(*

## Short summary
An abstract CycleManager implementation to provide basic functionality.
Does not update the state of the cyclemanager, it only provides some protected update functions.

.. <info>
If used in the same step, the order/precedence of method calls should be like this:
configurations
enter
executeCommand
evaluate
waitFor
proceed
proceedWith
acknowledge
leave
.. </info>

.. <legal notes>

legal notes
=================
| SPDX-FileCopyrightText: © 2024 ekvip automation GmbH <info@ekvip.de>
| SPDX-License-Identifier: Apache-2.0
| For details check: Apache-2.0_

.. _Apache-2.0: https://www.apache.org/licenses/LICENSE-2.0

.. </legal notes>



*)
FUNCTION_BLOCK ABSTRACT AbstractCycleManager 
EXTENDS CNM_AssertionInterfaces.AbstractAssertor 
IMPLEMENTS CNM_CycleManagerInterfaces.ISingleExecutionCycleManager, 
	CNM_CycleManagerInterfaces.ICycleManagerDefaultParameters, 
	ICycleManagerStepParameters
//config
VAR
	sequenceErrorStep :DINT := STEP_ERROR;
	sequencePauseEnabled :BOOL := FALSE;
	sequenceSteppingEnabled :BOOL := FALSE;
	sequenceTimeOut :TIME := T#0S;
	sequenceStopRequestMode :CNM_CycleManagerInterfaces.StepStopRequestMode := CNM_CycleManagerInterfaces.StepStopRequestMode.IGNORE;
	sequenceTimeoutStep :DINT := STEP_ERROR;
	sequenceStepWidth :DINT := 1;
	sequenceRequireSuccessStep :BOOL := FALSE;
	
	stepErrorStep :DINT := STEP_ERROR;
	stepPauseEnabled :BOOL := FALSE;
	stepSteppingEnabled :BOOL := FALSE;
	stepTimeOut :TIME := T#0S;
	stepCurrentStopRequestMode :CNM_CycleManagerInterfaces.StepStopRequestMode := CNM_CycleManagerInterfaces.StepStopRequestMode.IGNORE;
	stepTimeoutStep :DINT := STEP_ERROR;
	stepStepWidth :DINT := 1;
END_VAR
VAR
	lastStepBeforePause : DINT;
	lastStep : DINT;
	
	currentStep : DINT := CNM_ReturnTypes.DefaultSteps.STEP.IDLE;
	nextStep : DINT := CNM_ReturnTypes.DefaultSteps.STEP.IDLE;
	nextStepSpecifiedByUser :BOOL := FALSE;
	lastExecute : BOOL;
	externalExecute : BOOL;
	currentState : CNM_ReturnTypes.SingleExecutionState := CNM_ReturnTypes.SingleExecutionState.IDLE;
	wasError : BOOL;
	wasTimeoutError : BOOL;
	gotHereByError : BOOL;
	stepLastCycle : DINT;
	wasNotSuccess: BOOL;
	wasSuccess: BOOL;
	firstCycle : BOOL;
	timeoutTimer : TON;
	
	//used for cycle time optimizations
	registeredEnter : BOOL;
	registeredCommand : BOOL;
	registeredEval : BOOL;
	registeredLeave : BOOL;	
END_VAR
VAR CONSTANT
	STEP_IDLE :DINT := CNM_ReturnTypes.DefaultSteps.STEP.IDLE;
	STEP_INIT :DINT := CNM_ReturnTypes.DefaultSteps.STEP.INIT;
	STEP_ERROR :DINT := CNM_ReturnTypes.DefaultSteps.STEP.ERROR;
	STEP_ABORT :DINT := CNM_ReturnTypes.DefaultSteps.STEP.ABORT;
	STEP_PAUSE :DINT := CNM_ReturnTypes.DefaultSteps.STEP.PAUSE;
	STEP_SUCCESS :DINT := CNM_ReturnTypes.DefaultSteps.STEP.SUCCESS;	
END_VAR


(*

## Short summary
This method acknowledges an error in the state machine and resets the current step to the step befor the error occured.

.. <legal notes>

legal notes
=================
| SPDX-FileCopyrightText: © 2024 ekvip automation GmbH <info@ekvip.de>
| SPDX-License-Identifier: Apache-2.0
| For details check: Apache-2.0_

.. _Apache-2.0: https://www.apache.org/licenses/LICENSE-2.0

.. </legal notes>

*)
{attribute 'hide'}
METHOD acknowledge
IF(THIS^.gotHereByError)THEN
	THIS^.next := THIS^.last;
	THIS^.wasNotSuccess := FALSE;
	THIS^.wasError := FALSE;
	THIS^.wasTimeoutError := FALSE;
	THIS^.wasSuccess := TRUE;
END_IF
END_METHOD

(*

## Short summary
This method is called if an assertion was ``FALSE``

.. <legal notes>

legal notes
=================
| SPDX-FileCopyrightText: © 2022 ekvip automation GmbH <info@ekvip.de>
| SPDX-License-Identifier: Apache-2.0
| For details check: Apache-2.0_

.. _Apache-2.0: https://www.apache.org/licenses/LICENSE-2.0

.. </legal notes>


*)
METHOD assertionWasWrong
VAR_INPUT
	(* caller object of the method *)
	caller	: CNM_AbstractObject.IObject;
	(* alarm message *)
	message	: CNM_AssertionInterfaces.AssertMessage;
	(* debugging information *)
	additionalText	: Tc2_System.T_MaxString;
END_VAR
THIS^.wasError := TRUE;
THIS^.wasSuccess := FALSE;
THIS^.wasNotSuccess := TRUE;
END_METHOD

(*

## Short summary
An interface to provide configurations for cycle manager in a fluent way.

.. <legal notes>

legal notes
=================
| SPDX-FileCopyrightText: © 2024 ekvip automation GmbH <info@ekvip.de>
| SPDX-License-Identifier: Apache-2.0
| For details check: Apache-2.0_

.. _Apache-2.0: https://www.apache.org/licenses/LICENSE-2.0

.. </legal notes>



*)
PROPERTY configuration : CNM_CycleManagerInterfaces.ICycleManagerConfigurationScope
GET
VAR_INST
	configurator :CycleManagerConfigurator(THIS^, THIS^);
END_VAR
configuration := configurator;
END_GET
END_PROPERTY

(*

## Short summary
This property returns the current step of the cycle manager.
Proposed use is as CASE control.

### Example
```
CASE cyclemanager.steps.current OF
DefaultSteps.STEP.IDLE:
	;
DefaultSteps.STEP.INIT:
	;
2:
	;
3:
	;
4:
	;
DefaultSteps.STEP.SUCCESS:
	;
DefaultSteps.STEP.ERROR:
	;
DefaultSteps.STEP.ABORT:
	;
ELSE ;
END_CASE
```

.. <legal notes>

legal notes
=================
| SPDX-FileCopyrightText: © 2024 ekvip automation GmbH <info@ekvip.de>
| SPDX-License-Identifier: Apache-2.0
| For details check: Apache-2.0_

.. _Apache-2.0: https://www.apache.org/licenses/LICENSE-2.0

.. </legal notes>

*)
{attribute 'hide'}
PROPERTY current : DINT
GET
current := THIS^.currentStep;
END_GET
SET // PRIVATE
THIS^.currentStep := current;
END_SET
END_PROPERTY

{attribute 'hide'}
PROPERTY currentErrorStep : DINT
GET // PROTECTED
currentErrorStep := THIS^.stepErrorStep;
END_GET
SET
THIS^.stepErrorStep := currentErrorStep;
END_SET
END_PROPERTY

{attribute 'hide'}
PROPERTY currentPauseEnabled : BOOL
GET // PROTECTED
currentPauseEnabled := THIS^.stepPauseEnabled;
END_GET
SET
THIS^.stepPauseEnabled := currentPauseEnabled;
END_SET
END_PROPERTY

{attribute 'hide'}
PROPERTY currentSteppingEnabled : BOOL
GET // PROTECTED
currentSteppingEnabled := THIS^.stepSteppingEnabled;
END_GET
SET
THIS^.stepSteppingEnabled := currentSteppingEnabled;
END_SET
END_PROPERTY

{attribute 'hide'}
PROPERTY currentStepWidth : DINT
GET // PROTECTED
currentStepWidth := THIS^.stepStepWidth;
END_GET
SET
THIS^.stepStepWidth := currentStepWidth;
END_SET
END_PROPERTY

{attribute 'hide'}
PROPERTY currentStopRequestMode : CNM_CycleManagerInterfaces.StepStopRequestMode
GET // PROTECTED
currentStopRequestMode := THIS^.stepCurrentStopRequestMode;
END_GET
SET
THIS^.stepCurrentStopRequestMode := currentStopRequestMode;
END_SET
END_PROPERTY

(*

## Short summary
This property sets the maximum execution time for the current step. 
The cycle manager will go into the error step after the time elapsed.

.. <legal notes>

legal notes
=================
| SPDX-FileCopyrightText: © 2024 ekvip automation GmbH <info@ekvip.de>
| SPDX-License-Identifier: Apache-2.0
| For details check: Apache-2.0_

.. _Apache-2.0: https://www.apache.org/licenses/LICENSE-2.0

.. </legal notes>

*)
{attribute 'hide'}
PROPERTY currentTimeout : TIME
GET // PROTECTED
currentTimeout := THIS^.stepTimeOut;
END_GET
SET
THIS^.stepTimeOut := currentTimeout;
END_SET
END_PROPERTY

{attribute 'hide'}
PROPERTY currentTimeoutStep : DINT
GET // PROTECTED
IF(THIS^.stepTimeoutStep <> THIS^.defaultTimeoutStep OR THIS^.stepTimeoutStep <> THIS^.defaultErrorStep)THEN
	currentTimeoutStep := THIS^.stepTimeoutStep;	
ELSE
	currentTimeoutStep := THIS^.currentErrorStep;
END_IF
END_GET
SET
THIS^.stepTimeoutStep := currentTimeoutStep;
END_SET
END_PROPERTY

(*

## Short summary
This property stes the next step in case of an error after a step change.

.. <legal notes>

legal notes
=================
| SPDX-FileCopyrightText: © 2024 ekvip automation GmbH <info@ekvip.de>
| SPDX-License-Identifier: Apache-2.0
| For details check: Apache-2.0_

.. _Apache-2.0: https://www.apache.org/licenses/LICENSE-2.0

.. </legal notes>

*)

{attribute 'hide'}
PROPERTY defaultErrorStep : DINT
GET // PROTECTED
defaultErrorStep := THIS^.sequenceErrorStep;
END_GET
SET
THIS^.sequenceErrorStep := defaultErrorStep;
THIS^.currentErrorStep := defaultErrorStep;
END_SET
END_PROPERTY

(*

## Short summary
This property sets the default pause enabling state after a step change.

.. <legal notes>

legal notes
=================
| SPDX-FileCopyrightText: © 2024 ekvip automation GmbH <info@ekvip.de>
| SPDX-License-Identifier: Apache-2.0
| For details check: Apache-2.0_

.. _Apache-2.0: https://www.apache.org/licenses/LICENSE-2.0

.. </legal notes>

*)

{attribute 'hide'}
PROPERTY defaultPauseEnabled : BOOL
GET // PROTECTED
defaultPauseEnabled := THIS^.sequencePauseEnabled;
END_GET
SET
THIS^.sequencePauseEnabled := defaultPauseEnabled;
THIS^.currentPauseEnabled := defaultPauseEnabled;
END_SET
END_PROPERTY

(*

## Short summary
Specifies whether the SUCCESS step of the state machine can be skipped when the transition condition to SUCCESS is already fulfilled.

When set to false, the state machine immediately returns SUCCESS as soon as the transition condition to the SUCCESS state is met, 
without executing the dedicated SUCCESS step. This optimization can save one execution cycle per state machine invocation, which is 
especially beneficial in nested or complex state machine structures.

When set to true, the SUCCESS step will always be executed at least once before the state machine returns SUCCESS. This is required 
in cases where the SUCCESS step performs essential actions (e.g., resetting outputs, logging, or cleanup).

The default value is false.

Use Case:
Use false when the SUCCESS step has no functional side effects and skipping it can improve performance.
Use true when the SUCCESS step contains logic that must be executed explicitly.

.. <legal notes>

legal notes
=================
| SPDX-FileCopyrightText: © 2025 ekvip automation GmbH <info@ekvip.de>
| SPDX-License-Identifier: Apache-2.0
| For details check: Apache-2.0_

.. _Apache-2.0: https://www.apache.org/licenses/LICENSE-2.0

.. </legal notes>

*)

PROPERTY defaultRequireSuccessStep : BOOL
GET
defaultRequireSuccessStep := THIS^.sequenceRequireSuccessStep;
END_GET
SET
THIS^.sequenceRequireSuccessStep := defaultRequireSuccessStep;
END_SET
END_PROPERTY

(*

## Short summary
This property sets the default stepping mode configuration after a step change.

.. <legal notes>

legal notes
=================
| SPDX-FileCopyrightText: © 2024 ekvip automation GmbH <info@ekvip.de>
| SPDX-License-Identifier: Apache-2.0
| For details check: Apache-2.0_

.. _Apache-2.0: https://www.apache.org/licenses/LICENSE-2.0

.. </legal notes>

*)

{attribute 'hide'}
PROPERTY defaultSteppingEnabled : BOOL
GET // PROTECTED
defaultSteppingEnabled := THIS^.sequenceSteppingEnabled;
END_GET
SET
THIS^.sequenceSteppingEnabled := defaultSteppingEnabled;
THIS^.currentSteppingEnabled := defaultSteppingEnabled;
END_SET
END_PROPERTY

(*

## Short summary
This property sets the default the step width.

.. <legal notes>

legal notes
=================
| SPDX-FileCopyrightText: © 2024 ekvip automation GmbH <info@ekvip.de>
| SPDX-License-Identifier: Apache-2.0
| For details check: Apache-2.0_

.. _Apache-2.0: https://www.apache.org/licenses/LICENSE-2.0

.. </legal notes>

*)

{attribute 'hide'}
PROPERTY defaultStepWidth : DINT
GET // PROTECTED
defaultStepWidth := THIS^.sequenceStepWidth;
END_GET
SET
THIS^.sequenceStepWidth := defaultStepWidth;
THIS^.currentStepWidth := defaultStepWidth;
END_SET
END_PROPERTY

(*

## Short summary
This property sets the default step mode configuration. 

.. <legal notes>

legal notes
=================
| SPDX-FileCopyrightText: © 2024 ekvip automation GmbH <info@ekvip.de>
| SPDX-License-Identifier: Apache-2.0
| For details check: Apache-2.0_

.. _Apache-2.0: https://www.apache.org/licenses/LICENSE-2.0

.. </legal notes>

*)

{attribute 'hide'}
PROPERTY defaultStopRequestMode : CNM_CycleManagerInterfaces.StepStopRequestMode
GET // PROTECTED
defaultStopRequestMode := THIS^.sequenceStopRequestMode;
END_GET
SET
THIS^.sequenceStopRequestMode := defaultStopRequestMode;
THIS^.currentStopRequestMode := defaultStopRequestMode;
END_SET
END_PROPERTY

(*

## Short summary
This property sets the maximum execution time for steps. 
The cycle manager will go into the timeoutStep after the time elapsed.

.. <legal notes>

legal notes
=================
| SPDX-FileCopyrightText: © 2024 ekvip automation GmbH <info@ekvip.de>
| SPDX-License-Identifier: Apache-2.0
| For details check: Apache-2.0_

.. _Apache-2.0: https://www.apache.org/licenses/LICENSE-2.0

.. </legal notes>

*)

{attribute 'hide'}
PROPERTY defaultTimeout : TIME
GET // PROTECTED
defaultTimeout := THIS^.sequenceTimeOut;
END_GET
SET
THIS^.sequenceTimeOut := defaultTimeout;
THIS^.currentTimeout := defaultTimeout;
END_SET
END_PROPERTY

(*

## Short summary
This property sets the default step that will be set if the current step reaches a timeout. 

.. <legal notes>

legal notes
=================
| SPDX-FileCopyrightText: © 2024 ekvip automation GmbH <info@ekvip.de>
| SPDX-License-Identifier: Apache-2.0
| For details check: Apache-2.0_

.. _Apache-2.0: https://www.apache.org/licenses/LICENSE-2.0

.. </legal notes>

*)

{attribute 'hide'}
PROPERTY defaultTimeoutStep : DINT
GET // PROTECTED
defaultTimeoutStep := THIS^.sequenceTimeoutStep;
END_GET
SET
THIS^.sequenceTimeoutStep := defaultTimeoutStep;
THIS^.currentTimeoutStep := defaultTimeoutStep;
END_SET
END_PROPERTY

(*

## Short summary
This method performs the given invoke only in the first cycle of the current step.

.. <legal notes>

legal notes
=================
| SPDX-FileCopyrightText: © 2024 ekvip automation GmbH <info@ekvip.de>
| SPDX-License-Identifier: Apache-2.0
| For details check: Apache-2.0_

.. _Apache-2.0: https://www.apache.org/licenses/LICENSE-2.0

.. </legal notes>


*)
METHOD enter
VAR_INPUT
	(* command to execute *)
	invoke	:CNM_CommandInterfaces.ISingleAttempt;
	(* step to proceed with in case of error *)
	errorStep	:DINT := CNM_ReturnTypes.DefaultSteps.STEP.ERROR;
END_VAR
THIS^.registeredEnter := TRUE;

RETURN (
	THIS^.executeStep 
	OR_ELSE THIS^.state <> CNM_ReturnTypes.SingleExecutionState.BUSY
);

IF (THIS^.isObjectNull(invoke) OR_ELSE (invoke.invoke() <> CNM_ReturnTypes.SingleExecutionResult.SUCCESS)) THEN
	THIS^.wasError := TRUE;
	THIS^.wasSuccess := FALSE;
	IF ((errorStep <> CNM_ReturnTypes.DefaultSteps.STEP.ERROR) 
		AND_THEN (errorStep <> THIS^.currentErrorStep)
	) THEN
		THIS^.currentErrorStep := errorStep;
	END_IF
END_IF
END_METHOD

(*

## Short summary
This property returns an ``ICycleError`` interface fluently to provide error handling methods.

.. <legal notes>

legal notes
=================
| SPDX-FileCopyrightText: © 2024 ekvip automation GmbH <info@ekvip.de>
| SPDX-License-Identifier: Apache-2.0
| For details check: Apache-2.0_

.. _Apache-2.0: https://www.apache.org/licenses/LICENSE-2.0

.. </legal notes>

*)
PROPERTY errors : CNM_CycleManagerInterfaces.ICycleError
GET
errors := THIS^;
END_GET
END_PROPERTY

(*

## Short summary
This method evaluates an execution state to calculate the next step.

.. <legal notes>

legal notes
=================
| SPDX-FileCopyrightText: © 2024 ekvip automation GmbH <info@ekvip.de>
| SPDX-License-Identifier: Apache-2.0
| For details check: Apache-2.0_

.. _Apache-2.0: https://www.apache.org/licenses/LICENSE-2.0

.. </legal notes>

*)
METHOD evaluate
VAR_INPUT
	(* the state which is to be evaluated *)
	state	:CNM_ReturnTypes.SingleExecutionState;
	(* step to proceed with in case of error *)
	errorStep	:DINT := CNM_ReturnTypes.DefaultSteps.STEP.ERROR;
END_VAR
THIS^.registeredEval := TRUE;

RETURN ( 	
		THIS^.wasError 
	OR_ELSE 
		(THIS^.state <> CNM_ReturnTypes.SingleExecutionState.BUSY)
	OR_ELSE
		NOT THIS^.executeStep
);

CASE state OF
CNM_ReturnTypes.SingleExecutionState.ERROR, CNM_ReturnTypes.SingleExecutionState.ABORTED:
	THIS^.wasError := TRUE;
	THIS^.wasSuccess := FALSE;
	IF ((errorStep <> CNM_ReturnTypes.DefaultSteps.STEP.ERROR) 
		AND_THEN (errorStep <> THIS^.currentErrorStep)
	) THEN
		THIS^.currentErrorStep := errorStep;
	END_IF
CNM_ReturnTypes.SingleExecutionState.BUSY:
	THIS^.wasNotSuccess := TRUE;
	IF(NOT THIS^.wasError)THEN
		THIS^.wasSuccess := FALSE;
	END_IF
CNM_ReturnTypes.SingleExecutionState.SUCCESS:
	IF(NOT THIS^.wasError AND NOT THIS^.wasNotSuccess)THEN
		THIS^.wasSuccess := TRUE;	
	END_IF
CNM_ReturnTypes.SingleExecutionState.IDLE, CNM_ReturnTypes.SingleExecutionState.PAUSED:
	THIS^.wasNotSuccess := TRUE;
	IF(NOT THIS^.wasError)THEN
		THIS^.wasSuccess := FALSE;
	END_IF
END_CASE
END_METHOD

(*

## Short summary
This method performs the given command and evaluates the return value.
The command will be called with execute := FALSE in the first cylce and with execute := TRUE in all following

.. <legal notes>

legal notes
=================
| SPDX-FileCopyrightText: © 2024 ekvip automation GmbH <info@ekvip.de>
| SPDX-License-Identifier: Apache-2.0
| For details check: Apache-2.0_

.. _Apache-2.0: https://www.apache.org/licenses/LICENSE-2.0

.. </legal notes>

*)
METHOD executeCommand
VAR_INPUT
	(* command to execute *)
	command :CNM_CommandInterfaces.ICommand;
	(* step to proceed with in case of error *)
	errorStep :DINT := CNM_ReturnTypes.DefaultSteps.STEP.ERROR;
END_VAR
THIS^.registeredCommand := TRUE;

IF(THIS^.isObjectNull(command))THEN
	THIS^.evaluate(CNM_ReturnTypes.SingleExecutionState.ERROR, errorStep);	
ELSE
	THIS^.evaluate(command.executeCommand(THIS^.executeStep), errorStep);	
END_IF
END_METHOD

(*

## Short summary
This property returns the execute flag for the current step, 
which is FALSE in the first cycle of each step and TRUE after.

.. <legal notes>

legal notes
=================
| SPDX-FileCopyrightText: © 2024 ekvip automation GmbH <info@ekvip.de>
| SPDX-License-Identifier: Apache-2.0
| For details check: Apache-2.0_

.. _Apache-2.0: https://www.apache.org/licenses/LICENSE-2.0

.. </legal notes>

*)
PROPERTY executeStep :BOOL
GET
executeStep := THIS^.externalExecute;
END_GET
END_PROPERTY

METHOD PROTECTED getStateFromStep : CNM_ReturnTypes.SingleExecutionState
VAR_INPUT
	step :DINT;
END_VAR
CASE step OF
STEP_ABORT:
	getStateFromStep := CNM_ReturnTypes.SingleExecutionState.ABORTED;
STEP_ERROR:
	getStateFromStep := CNM_ReturnTypes.SingleExecutionState.ERROR;
STEP_PAUSE:
	getStateFromStep := CNM_ReturnTypes.SingleExecutionState.PAUSED;
STEP_SUCCESS:
	getStateFromStep := CNM_ReturnTypes.SingleExecutionState.SUCCESS;
STEP_IDLE:
	;
STEP_INIT:
	getStateFromStep := CNM_ReturnTypes.SingleExecutionState.BUSY;
ELSE
	//sequence is running
	getStateFromStep := CNM_ReturnTypes.SingleExecutionState.BUSY;
END_CASE
END_METHOD

(*

## Short summary
This method throws an alarm and waits for it to be confirmed. 
When the alarm was confirmed the cyclemanager will proceed to next configured step.
If the current step is the result of an evaulated error state and the input 'resumeWithLastStep' is set to true, the cyclemanager will proceed to the last step.
..warning:  The 'resumeWithLastStep' flag will be ignored if the last step was successful.

.. <legal notes>

legal notes
=================
| SPDX-FileCopyrightText: © 2024 ekvip automation GmbH <info@ekvip.de>
| SPDX-License-Identifier: Apache-2.0
| For details check: Apache-2.0_

.. _Apache-2.0: https://www.apache.org/licenses/LICENSE-2.0

.. </legal notes>

*)

METHOD handle
VAR_INPUT
	(* the alarm event that should be thrown *)
	alarm :CNM_MessageInterfaces.IAlarm;
	(* if this flag is set AND we got to the current step because of an ERROR state, then the cyclemanager will automatically will go back to the last step *)
	resumeWithLastStep :BOOL := TRUE;
END_VAR
IF(NOT THIS^.executeStep)THEN
	alarm.throw();
ELSIF(NOT alarm.isPending)THEN
	IF(resumeWithLastStep AND_THEN THIS^.gotHereByError)THEN
		THIS^.acknowledge();
	ELSE
		THIS^.evaluate(state := CNM_ReturnTypes.SingleExecutionState.SUCCESS);
	END_IF
END_IF
END_METHOD

(*

## Short summary
This method handles the resume function of the cycle manager.
Should be called befor all other handles.

.. <legal notes>

legal notes
=================
| SPDX-FileCopyrightText: © 2024 ekvip automation GmbH <info@ekvip.de>
| SPDX-License-Identifier: Apache-2.0
| For details check: Apache-2.0_

.. _Apache-2.0: https://www.apache.org/licenses/LICENSE-2.0

.. </legal notes>

*)
METHOD PROTECTED handleCycleManagerError
VAR_INPUT
	(*if true, will acknowledge error and return to previous step*)
	resume :BOOL;
END_VAR
IF(resume)THEN
	THIS^.acknowledge();
END_IF
END_METHOD

(*

## Short summary
This method handles the execution of the cycle manager.
Should be the first thing to do at the start of each cycle.

.. <legal notes>

legal notes
=================
| SPDX-FileCopyrightText: © 2024 ekvip automation GmbH <info@ekvip.de>
| SPDX-License-Identifier: Apache-2.0
| For details check: Apache-2.0_

.. _Apache-2.0: https://www.apache.org/licenses/LICENSE-2.0

.. </legal notes>

*)
METHOD PROTECTED handleCycleManagerExecute : BOOL
VAR_INPUT
	(*control bit to start or abort the cycle manager*)
	execute :BOOL;
END_VAR
IF(THIS^.lastExecute <> execute)THEN
	IF(execute)THEN
		//first cylce / init
		THIS^.currentState := CNM_ReturnTypes.SingleExecutionState.BUSY;
		THIS^.step.next := STEP_INIT;
		THIS^.firstCycle := TRUE;
	ELSE		
		//falling execute / reset
		IF(THIS^.currentState = CNM_ReturnTypes.SingleExecutionState.BUSY OR THIS^.currentState = CNM_ReturnTypes.SingleExecutionState.PAUSED)THEN
			THIS^.currentState := CNM_ReturnTypes.SingleExecutionState.ABORTED;
			THIS^.currentStep := STEP_ABORT;
		ELSE
			THIS^.currentStep := STEP_IDLE;	
			THIS^.step.next := STEP_IDLE;	
			THIS^.lastStep := STEP_IDLE;			
		END_IF
		THIS^.externalExecute := FALSE;
	END_IF
ELSIF(THIS^.currentStep = STEP_ABORT)THEN
	//only one cycle in ABORT Step
	THIS^.currentStep := STEP_IDLE;
END_IF

THIS^.lastExecute := execute;

handleCycleManagerExecute := execute;
END_METHOD

(*

## Short summary
This method handles the pausing of the cycle manager. 
Should be handled before updating.

.. <legal notes>

legal notes
=================
| SPDX-FileCopyrightText: © 2024 ekvip automation GmbH <info@ekvip.de>
| SPDX-License-Identifier: Apache-2.0
| For details check: Apache-2.0_

.. _Apache-2.0: https://www.apache.org/licenses/LICENSE-2.0

.. </legal notes>

*)
METHOD PROTECTED handleCycleManagerPause
VAR_INPUT
	(*if true and Pausing Enabled and busy will proceed with PAUSE*)
	pause :BOOL;
END_VAR
IF(NOT pause AND_THEN THIS^.currentState = CNM_ReturnTypes.SingleExecutionState.PAUSED)THEN
	THIS^.currentStep := THIS^.lastStepBeforePause;
END_IF

RETURN (NOT THIS^.currentPauseEnabled);

IF(
	pause 
	AND_THEN (NOT THIS^.wasError) 
	AND_THEN (THIS^.currentState = CNM_ReturnTypes.SingleExecutionState.BUSY)
)THEN
	THIS^.lastStepBeforePause := THIS^.currentStep;
	THIS^.currentStep := STEP_PAUSE;
END_IF
END_METHOD

(*

## Short summary
This method handles the timeout of the current step.
Call at any point each cycle.
.. <legal notes>

legal notes
=================
| SPDX-FileCopyrightText: © 2024 ekvip automation GmbH <info@ekvip.de>
| SPDX-License-Identifier: Apache-2.0
| For details check: Apache-2.0_

.. _Apache-2.0: https://www.apache.org/licenses/LICENSE-2.0

.. </legal notes>

*)
METHOD PROTECTED handleCycleManagerTimeout : BOOL
VAR_INPUT
	(* must be TRUE if stepping is enabled to proceed steps automatically *)
	step :BOOL;
END_VAR
IF ((THIS^.currentState = CNM_ReturnTypes.SingleExecutionState.BUSY) AND (THIS^.currentTimeout > T#0S)) THEN
	THIS^.timeoutTimer(
		IN := (
			(NOT THIS^.currentSteppingEnabled) 
			OR 
			(NOT step)
		), 
		PT := THIS^.currentTimeout,
		Q => THIS^.wasTimeoutError
	);
END_IF
END_METHOD

(*

## Short summary
This method handles the step change, call early in handling.

.. <legal notes>

legal notes
=================
| SPDX-FileCopyrightText: © 2024 ekvip automation GmbH <info@ekvip.de>
| SPDX-License-Identifier: Apache-2.0
| For details check: Apache-2.0_

.. _Apache-2.0: https://www.apache.org/licenses/LICENSE-2.0

.. </legal notes>

*)
METHOD PROTECTED handleStepChange
VAR_INPUT
	(* must be TRUE if stepping is enabled to proceed steps automatically *)
	step :BOOL := TRUE;
	(*used for StopRequest evaluation if configured*)
	stopRequest :BOOL := FALSE;
END_VAR
IF THIS^.wasError THEN
    THIS^.step.next := THIS^.currentErrorStep;
    THIS^.initializeNewStep(TRUE);

ELSIF THIS^.wasTimeoutError THEN
    THIS^.step.next := THIS^.currentTimeoutStep;
    THIS^.initializeNewStep(TRUE);

ELSIF stopRequest AND (
        (THIS^.wasSuccess AND NOT THIS^.wasNotSuccess AND (THIS^.executeStep OR NOT THIS^.isAnyActionRegistered)
            AND THIS^.currentStopRequestMode = CNM_CycleManagerInterfaces.StepStopRequestMode.AFTER_SUCCESSFUL_STEP)
     OR (THIS^.wasNotSuccess AND (THIS^.executeStep OR NOT THIS^.isAnyActionRegistered)
            AND THIS^.currentStopRequestMode = CNM_CycleManagerInterfaces.StepStopRequestMode.ON_BUSY)
     OR (THIS^.currentStopRequestMode = CNM_CycleManagerInterfaces.StepStopRequestMode.IMMEDIATE)
) THEN
    THIS^.step.next := STEP_SUCCESS;
    THIS^.initializeNewStep();

ELSIF THIS^.wasSuccess
	AND NOT THIS^.wasNotSuccess 
	AND (THIS^.executeStep OR NOT THIS^.isAnyActionRegistered)
    AND (NOT THIS^.currentSteppingEnabled OR step) 
THEN
    THIS^.initializeNewStep();
END_IF
END_METHOD

METHOD PRIVATE initializeNewStep
VAR_INPUT
	errorStep :BOOL := FALSE;
END_VAR
THIS^.gotHereByError := errorStep;
THIS^.firstCycle := TRUE;
END_METHOD

(*

## Short summary
This boolean is true when at least one of these actions are registered:
- executeCommand
- evaluate
- leave

The setter can be used to clear all the registered actions at once. 

.. <legal notes>

legal notes
=================
| SPDX-FileCopyrightText: © 2025 ekvip automation GmbH <info@ekvip.de>
| SPDX-License-Identifier: Apache-2.0
| For details check: Apache-2.0_

.. _Apache-2.0: https://www.apache.org/licenses/LICENSE-2.0

.. </legal notes>

*)

PROPERTY PROTECTED isAnyActionRegistered : BOOL
GET
isAnyActionRegistered := THIS^.registeredCommand OR THIS^.registeredLeave OR THIS^.registeredEval;
END_GET
SET
RETURN(isAnyActionRegistered); //dont set all the flags to true at once
THIS^.registeredCommand := 
THIS^.registeredEval := 
THIS^.registeredLeave := isAnyActionRegistered; // only if isAnyActionRegistered is set to false
END_SET
END_PROPERTY

(*

## Short summary
This property returns TRUE if the step was reached by evaluating an error.

.. <legal notes>

legal notes
=================
| SPDX-FileCopyrightText: © 2024 ekvip automation GmbH <info@ekvip.de>
| SPDX-License-Identifier: Apache-2.0
| For details check: Apache-2.0_

.. _Apache-2.0: https://www.apache.org/licenses/LICENSE-2.0

.. </legal notes>

*)
{attribute 'hide'}
PROPERTY isInErrorStep :BOOL
GET
isInErrorStep := THIS^.gotHereByError;
END_GET
END_PROPERTY

(*

## Short summary
This property returns the last step of the cycle manager, useful for error steps.

.. <legal notes>

legal notes
=================
| SPDX-FileCopyrightText: © 2024 ekvip automation GmbH <info@ekvip.de>
| SPDX-License-Identifier: Apache-2.0
| For details check: Apache-2.0_

.. _Apache-2.0: https://www.apache.org/licenses/LICENSE-2.0

.. </legal notes>

### Example
```
TIMEOUT_STEP_FOR_RETRY:
	cM.steps.next := cM.steps.last-1;
	cM.waitFor(ACK);

*)
{attribute 'hide'}
PROPERTY last : DINT
GET
last := SEL(THIS^.currentStep = STEP_PAUSE, THIS^.lastStep, THIS^.lastStepBeforePause);
END_GET
SET // PROTECTED
THIS^.lastStep := last;
END_SET
END_PROPERTY

(*

## Short summary
This method performs the given invoke only in the last cycle of the current step.

.. <legal notes>

legal notes
=================
| SPDX-FileCopyrightText: © 2024 ekvip automation GmbH <info@ekvip.de>
| SPDX-License-Identifier: Apache-2.0
| For details check: Apache-2.0_

.. _Apache-2.0: https://www.apache.org/licenses/LICENSE-2.0

.. </legal notes>

*)
METHOD leave
VAR_INPUT
	(* command to execute *)
	invoke	:CNM_CommandInterfaces.ISingleAttempt;
	(* step to proceed with in case of error *)
	errorStep	:DINT := CNM_ReturnTypes.DefaultSteps.STEP.ERROR; 
	(* whether the invoke should be called even if there was an error in the current step *)
	forceOnError	:BOOL := FALSE;
END_VAR
THIS^.registeredLeave := TRUE;

RETURN ((
			((NOT wasSuccess) OR_ELSE THIS^.wasNotSuccess) 
		AND 
			NOT(forceOnError AND THIS^.wasError)
		) 
	OR 
		THIS^.state <> CNM_ReturnTypes.SingleExecutionState.BUSY
);

IF(THIS^.isObjectNull(invoke) OR_ELSE invoke.invoke() <> CNM_ReturnTypes.SingleExecutionResult.SUCCESS)THEN
	THIS^.evaluate(CNM_ReturnTypes.SingleExecutionState.ERROR, errorStep);	
END_IF
END_METHOD

(*

## Short summary
This property sets the next step of the cycle manager.

.. <legal notes>

legal notes
=================
| SPDX-FileCopyrightText: © 2024 ekvip automation GmbH <info@ekvip.de>
| SPDX-License-Identifier: Apache-2.0
| For details check: Apache-2.0_

.. _Apache-2.0: https://www.apache.org/licenses/LICENSE-2.0

.. </legal notes>

### Example
```
MY_STEP:
	cyclemanager.steps.next := SUCCESS_STEP;
	cyclemanager.executeCommand(finalizeProcess);
	
*)
{attribute 'hide'}
PROPERTY next : DINT
GET
next := SEL(THIS^.nextStepSpecifiedByUser, THIS^.currentStep + THIS^.currentStepWidth, THIS^.nextStep);
END_GET
SET
THIS^.nextStep := next;
THIS^.nextStepSpecifiedByUser := TRUE;
END_SET
END_PROPERTY

(*

## Short summary
This method changes the current step in the cycle manager to the next in order (current + stepWidth) .
If any evaluate or other call is still busy it will ignore them and change to the next step.

.. <legal notes>

legal notes
=================
| SPDX-FileCopyrightText: © 2024 ekvip automation GmbH <info@ekvip.de>
| SPDX-License-Identifier: Apache-2.0
| For details check: Apache-2.0_

.. _Apache-2.0: https://www.apache.org/licenses/LICENSE-2.0

.. </legal notes>

*)
METHOD proceed
RETURN (THIS^.state = CNM_ReturnTypes.SingleExecutionState.SUCCESS);

THIS^.wasNotSuccess := FALSE;
THIS^.wasSuccess := TRUE;
THIS^.isAnyActionRegistered := FALSE;
END_METHOD

(*

## Short summary
This method changes the current step in the cycle manager to the given step.
If any evaluate or other call is still busy it will ignore them and move to the next step.

.. <legal notes>

legal notes
=================
| SPDX-FileCopyrightText: © 2024 ekvip automation GmbH <info@ekvip.de>
| SPDX-License-Identifier: Apache-2.0
| For details check: Apache-2.0_

.. _Apache-2.0: https://www.apache.org/licenses/LICENSE-2.0

.. </legal notes>

*)
METHOD proceedWith
VAR_INPUT
	(* step to move to *)
	step	:DINT;
END_VAR
RETURN (THIS^.state = CNM_ReturnTypes.SingleExecutionState.SUCCESS);

THIS^.step.next := step;
THIS^.proceed();
END_METHOD

METHOD PROTECTED resetCurrentStepParametersToDefaults
VAR_INPUT
END_VAR
THIS^.currentErrorStep := THIS^.defaultErrorStep;
THIS^.currentPauseEnabled := THIS^.defaultPauseEnabled;
THIS^.currentSteppingEnabled := THIS^.defaultSteppingEnabled;
THIS^.currentStepWidth := THIS^.defaultStepWidth;
THIS^.currentStopRequestMode := THIS^.defaultStopRequestMode;
THIS^.currentTimeoutStep := THIS^.defaultTimeoutStep;
THIS^.currentTimeout := THIS^.defaultTimeout;
END_METHOD

METHOD PROTECTED resetInternalVariables
THIS^.registeredCommand := FALSE;
THIS^.registeredEnter := FALSE;
THIS^.registeredEval := FALSE;
THIS^.registeredLeave := FALSE;	
THIS^.wasError := FALSE;
THIS^.wasTimeoutError := FALSE;
THIS^.wasNotSuccess := FALSE;
THIS^.wasSuccess := FALSE;
THIS^.firstCycle := FALSE;
THIS^.nextStepSpecifiedByUser := FALSE;
END_METHOD

(*

## Short summary
This property returns the current state of the cycle manager according to its step.

.. <legal notes>

legal notes
=================
| SPDX-FileCopyrightText: © 2024 ekvip automation GmbH <info@ekvip.de>
| SPDX-License-Identifier: Apache-2.0
| For details check: Apache-2.0_

.. _Apache-2.0: https://www.apache.org/licenses/LICENSE-2.0

.. </legal notes>

*)
PROPERTY state : CNM_ReturnTypes.SingleExecutionState
GET
VAR CONSTANT
	WAITING : DINT := 42;
END_VAR
IF(
	NOT THIS^.sequenceRequireSuccessStep
	AND_THEN NOT THIS^.wasError 
	AND_THEN wasSuccess 
	AND_THEN (THIS^.executeStep OR NOT(THIS^.registeredEval OR THIS^.registeredCommand OR THIS^.registeredLeave))
	AND_THEN THIS^.step.next = STEP_SUCCESS
)THEN
	//this allows the cycle manager to return SUCCESS one cycle earlier, saving many cycles in nested use
	THIS^.currentState := CNM_ReturnTypes.SingleExecutionState.SUCCESS;
END_IF

state := THIS^.currentState;
END_GET
SET // PROTECTED
THIS^.currentState := state;
END_SET
END_PROPERTY

(*

## Short summary
This property returns the current, next and last step of the cycle manager via fluent interface with the ``ICylceSteps`` interfaces

.. <legal notes>

legal notes
=================
| SPDX-FileCopyrightText: © 2024 ekvip automation GmbH <info@ekvip.de>
| SPDX-License-Identifier: Apache-2.0
| For details check: Apache-2.0_

.. _Apache-2.0: https://www.apache.org/licenses/LICENSE-2.0

.. </legal notes>

*)
PROPERTY step : CNM_CycleManagerInterfaces.ICycleSteps
GET
step := THIS^;
END_GET
END_PROPERTY

(*

## Short summary
This method handles all updates of the cycle manager.
Should be called first each cycle befor evaluating the steps and only once per cycle!

.. <legal notes>

legal notes
=================
| SPDX-FileCopyrightText: © 2024 ekvip automation GmbH <info@ekvip.de>
| SPDX-License-Identifier: Apache-2.0
| For details check: Apache-2.0_

.. _Apache-2.0: https://www.apache.org/licenses/LICENSE-2.0

.. </legal notes>

*)
METHOD update
VAR_INPUT
	(*control bit to start or abort the cycle manager*)
	execute :BOOL;
	(*used for StopRequest evaluation if configured*)
	stopRequest :BOOL := FALSE;
	(*if true and Pausing Enabled and busy will proceed with PAUSE*)
	pause :BOOL := FALSE;
	(*if true, will acknowledge error and return to previous step*)
	resume :BOOL := FALSE;
	(* must be TRUE if stepping is enabled to proceed steps automatically *)
	stepControl :BOOL := TRUE;
END_VAR
RETURN (NOT THIS^.handleCycleManagerExecute(execute));
THIS^.handleCycleManagerError(resume);
THIS^.handleStepChange(stepControl, stopRequest);
THIS^.handleCycleManagerPause(pause);
THIS^.handleCycleManagerTimeout(stepControl);
THIS^.updateCycleManager();
END_METHOD

(*

## Short summary
This method updates the step and state of the cycle manager.
Should be called after all handles each cycle.

.. <legal notes>

legal notes
=================
| SPDX-FileCopyrightText: © 2024 ekvip automation GmbH <info@ekvip.de>
| SPDX-License-Identifier: Apache-2.0
| For details check: Apache-2.0_

.. _Apache-2.0: https://www.apache.org/licenses/LICENSE-2.0

.. </legal notes>

*)
METHOD PROTECTED updateCycleManager
THIS^.externalExecute := NOT THIS^.firstCycle;

IF (THIS^.firstCycle AND_THEN (THIS^.currentStep <> CNM_ReturnTypes.DefaultSteps.STEP.SUCCESS)) THEN
	THIS^.timeoutTimer(IN := FALSE);
	
	THIS^.last := THIS^.currentStep;
	THIS^.currentStep := THIS^.step.next;
	
	THIS^.resetInternalVariables();
	THIS^.resetCurrentStepParametersToDefaults();
END_IF

//Set State for external use
THIS^.state := getStateFromStep(THIS^.currentStep);

THIS^.wasError := FALSE;
THIS^.wasNotSuccess := FALSE;
THIS^.wasSuccess := FALSE;
END_METHOD

(*

## Short summary
This method waits for a boolean signal until the step can be changed. 

.. <legal notes>

legal notes
=================
| SPDX-FileCopyrightText: © 2024 ekvip automation GmbH <info@ekvip.de>
| SPDX-License-Identifier: Apache-2.0
| For details check: Apache-2.0_

.. _Apache-2.0: https://www.apache.org/licenses/LICENSE-2.0

.. </legal notes>

*)
METHOD waitFor
VAR_INPUT
	(* the value to wait for *)
	value	:BOOL;
END_VAR
RETURN (THIS^.state <> CNM_ReturnTypes.SingleExecutionState.BUSY);

THIS^.registeredEval := TRUE;

IF(value)THEN
	IF(NOT wasError)THEN
		THIS^.wasSuccess := TRUE;
	END_IF
ELSE
	THIS^.wasNotSuccess := TRUE;
END_IF
END_METHOD

END_FUNCTION_BLOCK

(* stored: Version 1.1.0.1
   POU AbstractCycleManager: Id {2a2c30e9-a800-4b85-ab85-c34497491877}, SpecialFunc None
   Folder Assertor: Id {6508dab8-9ad3-449e-90d2-f33e17e2f23d}
   Folder config: Id {f7fe6a56-060e-4052-94ac-4806875d6a95}
   Folder defaults: Id {49365529-45b0-4d6d-a4c5-427847fec121}
   Folder step: Id {044518e2-1fa3-415e-b6d5-f011d33af915}
   Folder Errors: Id {8b8fa45c-af98-4dd6-bf05-e7112a5147d8}
   Folder ICycleManager: Id {3a2bf34f-0f10-4eca-9272-1dd595d51eac}
   Folder protected: Id {ee216269-00ac-48f7-8f6b-6de74dd3d5a3}
   Folder Steps: Id {9219762d-50a8-47cc-88eb-492ea15ae3ec}
   Method acknowledge: Id {3eca993e-8530-4fc4-ba48-3013af35c775}
   Method assertionWasWrong: Id {be71953c-ed01-49f3-aec2-0193acc08101}
   Property configuration: Id {38eee25d-ee93-42a6-83ca-edd29c7eba04}
   Get Get: Id {9c2ee367-d7f1-4cc2-ba2a-996913677975}
   Property current: Id {86a9da60-7c51-47c2-a053-c19947f9f9ee}
   Get Get: Id {bddaedd0-c1bc-4fe3-a2a0-04abda65c439}
   Set Set: Id {6fb55603-bc19-47d0-ae3b-28d64d07a8bc}
   Property currentErrorStep: Id {0c9e38b0-c14c-4cc9-8a36-320dff8392b3}
   Get Get: Id {5364b894-6ab1-4369-90a5-141d0ea398a6}
   Set Set: Id {fde72ff1-cb74-4100-9ead-9de98c06489e}
   Property currentPauseEnabled: Id {ce2e0c47-2eac-4a5d-ba31-e8745f720110}
   Get Get: Id {cf3ab530-fcad-4e0f-a37e-aff37489b461}
   Set Set: Id {55e2aabe-fc5e-40e9-8339-e981013e9579}
   Property currentSteppingEnabled: Id {9eabf085-2941-466f-b844-98b7df31229d}
   Get Get: Id {66cb4fce-8f59-4033-8ef5-a8ba3848c2cd}
   Set Set: Id {2deab1a0-4865-47e5-8226-e784e7b47083}
   Property currentStepWidth: Id {ad8c25db-02e6-4942-894a-55bb5f90decf}
   Get Get: Id {816c9ac8-c259-461f-8ad9-e29de5f8cbed}
   Set Set: Id {56e4ab57-74bd-4e90-8e29-1cd206fd4e76}
   Property currentStopRequestMode: Id {e4a37bb8-b1aa-427d-9899-8fb04b4c8465}
   Get Get: Id {ac13af56-d8bd-44ab-9111-f9bdc365ded2}
   Set Set: Id {5933b7d2-33fe-40b0-ba60-fab6c5176c4b}
   Property currentTimeout: Id {144a5160-4a45-490d-b795-abbda164aaf7}
   Get Get: Id {bbb99ba0-a0cb-4e83-84ba-43bc7df02fd4}
   Set Set: Id {de5f18dd-6ac1-423a-b489-bc31394793d3}
   Property currentTimeoutStep: Id {1c3d0f5a-90a4-4fb7-9e1b-0983aec59dc6}
   Get Get: Id {c66b0f21-7ba3-48a6-adde-c59b70313eba}
   Set Set: Id {a2e050a3-5893-488f-9221-308a970d656e}
   Property defaultErrorStep: Id {d69e7961-2f16-4b89-976c-b9177a5dcd1e}
   Get Get: Id {508803c8-2157-45ed-9c05-743ddde8631a}
   Set Set: Id {2445a279-98ba-4f53-84db-8eafb9cd3fd6}
   Property defaultPauseEnabled: Id {f3b3b0ab-0b3a-4287-a131-2dc0aa052a58}
   Get Get: Id {b15b9da6-fe4f-428b-b978-129bfbef0bb9}
   Set Set: Id {e4704ad1-7510-45b1-9736-d11005e4ce9c}
   Property defaultRequireSuccessStep: Id {8f83c82e-3913-4628-adf9-77eb77c7a712}
   Get Get: Id {7c3261aa-bc40-47d1-bb45-a7e1b859164e}
   Set Set: Id {f0e454ba-7b2e-426d-b4c4-7e71d9cb4aae}
   Property defaultSteppingEnabled: Id {c77a62c3-6663-4ce6-b624-031edaa021ff}
   Get Get: Id {ffb52f98-fac0-454f-8e9b-ad69c8af8db9}
   Set Set: Id {38cbbdfd-0f81-4eb7-8443-63a4d65280a9}
   Property defaultStepWidth: Id {44145af9-05fd-4a74-b6f9-61c1f8a8244c}
   Get Get: Id {b7edb333-0661-4f32-bd25-fd743dec49a8}
   Set Set: Id {87397639-afef-45ca-b560-57f26be1545e}
   Property defaultStopRequestMode: Id {777ac0fe-ab7d-4b41-aad8-f3b580999ada}
   Get Get: Id {c7e98599-e324-4a21-b765-5d64814aa25e}
   Set Set: Id {f2c4c467-297f-4ce2-b577-3ace13505151}
   Property defaultTimeout: Id {30c59382-a003-425c-b50a-2af7dbff6b6b}
   Get Get: Id {28e139d1-a253-44f0-bf93-cc8a9b116b92}
   Set Set: Id {02e5b274-457d-46f1-a829-46b9d60f15c0}
   Property defaultTimeoutStep: Id {08bb7765-1d12-4c7e-8c78-618de981c5a5}
   Get Get: Id {e42bc9b1-335e-4170-9d43-d1d43b7a51cb}
   Set Set: Id {d3650711-9c4a-4609-8724-d0ab55292f70}
   Method enter: Id {28872812-5eff-4b54-aaf6-4ce28b1e1b62}
   Property errors: Id {cbf9c447-4041-4d3b-81c2-0690657df719}
   Get Get: Id {ea2a1517-0df9-4ac5-9f2a-5f3c4139ab7f}
   Method evaluate: Id {8014ce81-4505-41cb-ad22-a1981d8bd067}
   Method executeCommand: Id {fe2a6303-5dcf-4215-ba88-018fff946858}
   Property executeStep: Id {1459dc10-209b-423f-8074-b703a90ef3cf}
   Get Get: Id {c9c8eb8b-bacd-496a-98db-8798ed14e3ec}
   Method getStateFromStep: Id {af81cd18-3e62-4700-a94a-f7098d846d5c}
   Method handle: Id {fb4d3ddc-45bb-4a27-81f7-5bcbed05db77}
   Method handleCycleManagerError: Id {8165ad7e-5581-4ba6-9059-5ac24957aa48}
   Method handleCycleManagerExecute: Id {530db549-ace4-41c5-92e2-755b05b5931f}
   Method handleCycleManagerPause: Id {c12329da-33c5-4eed-91d4-8486e78973af}
   Method handleCycleManagerTimeout: Id {bbc66314-ae57-4c95-897a-4df3555110b4}
   Method handleStepChange: Id {f418734f-3339-4477-a561-a0ee24a7824b}
   Method initializeNewStep: Id {ff926e09-08d2-4640-89c2-6d4d0dbc7c25}
   Property isAnyActionRegistered: Id {8dd98195-cf2b-4074-832d-21d519c3b662}
   Get Get: Id {3c33e752-fd46-4e6b-b2a1-0b56d3f20f78}
   Set Set: Id {3eee91a2-2eab-4ed9-8d78-1ec5e459aa7c}
   Property isInErrorStep: Id {9f42069f-c2f6-4cfc-aef9-100c905f26ea}
   Get Get: Id {b35899f0-2d63-411f-820f-e558909bd019}
   Property last: Id {f1d14b8b-7243-4122-9776-7df92fa6498e}
   Get Get: Id {4a5e142a-95d9-46c9-ae5f-89e921548a7f}
   Set Set: Id {a391eafb-7a2b-44c2-8304-53b4610ada5e}
   Method leave: Id {d1695d08-e2b2-48f6-91ef-52cd8438e2bb}
   Property next: Id {c1d03f67-dd21-4b2a-9788-84323d0761da}
   Get Get: Id {7f8c4a03-12c8-4693-a2b7-acb5a025de59}
   Set Set: Id {fb42c9c9-4095-45d5-b6c1-371b4d79a887}
   Method proceed: Id {0518105d-d4cd-4fe9-ad2e-ecb16b85e6f7}
   Method proceedWith: Id {1b4d17c5-2ec7-4cc4-bbcf-0a151536b5c2}
   Method resetCurrentStepParametersToDefaults: Id {f877d5bb-f145-465e-aeda-6e88b39304db}
   Method resetInternalVariables: Id {fef106fe-382a-4c28-b2f0-eac600379abd}
   Property state: Id {e7969c8f-f4bd-46dc-838c-23ae907bf0dd}
   Get Get: Id {51cad091-e8c1-478f-96f2-f5ef8397a3c3}
   Set Set: Id {13e49b80-7825-4d13-b384-9ac369628d5a}
   Property step: Id {7be67d05-dc27-4718-8761-9c0cb420c090}
   Get Get: Id {9709475d-1451-470e-8a2e-88fb5a8d28d5}
   Method update: Id {f3ca0071-adf4-4c4c-8551-be8f6724073e}
   Method updateCycleManager: Id {5938120f-5baa-41df-857f-38759da8e975}
   Method waitFor: Id {3544ee7e-949d-4b9b-baf9-ff9da311526c} *)
